FUNCTION_BLOCK PY_MQTT_SUB (* Basic FB with empty ECC *)
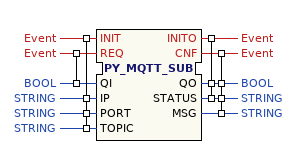
  EVENT_INPUT
    INIT WITH PORT, TOPIC, IP;
    REQ WITH QI;
  END_EVENT
  EVENT_OUTPUT
    INITO WITH QO, STATUS;
    CNF WITH MSG, STATUS, QO;
  END_EVENT
  VAR_INPUT
    QI : BOOL;
    IP : STRING;
    PORT : STRING;
    TOPIC : STRING;
  END_VAR
  VAR_OUTPUT
    QO : BOOL;
    STATUS : STRING;
    MSG : STRING;
  END_VAR
END_FUNCTION_BLOCK
